PROGRAM PRG_LD


VAR
    // 数据表格式
 

    // 连接到数据库
 

    // 插入新行
 

    // 查询现有数据
 

    // 更新现有数据
 


stTableSchema        : ST_ProdColumnName;;

FB_ConnSQLServer_0   : FB_ConnSQLServer;;

stNewProd            : ST_ProdEntry;;

FB_InsertSQLServer_0 : FB_InsertSQLServer;;

stQueryProd          : ST_ProdEntry;;

FB_QuerySQLServer_0  : FB_QuerySQLServer;;

stUpdateProd         : ST_ProdEntry;;

FB_UpdateSQLServer_0 : FB_UpdateSQLServer;;

    END_VAR

END_PROGRAM

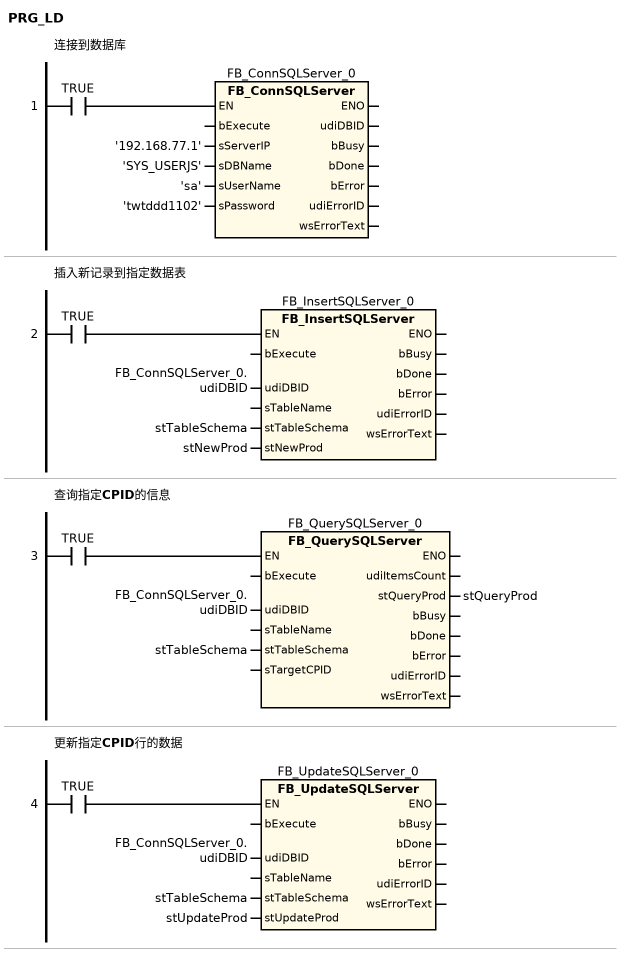
// NETWORK 1: 连接到数据库
FB_ConnSQLServer_0(
    sServerIP := '192.168.77.1',
    sDBName := 'SYS_USERJS',
    sUserName := 'sa',
    sPassword := 'twtddd1102'); // FB_ConnSQLServer

// NETWORK 2: 插入新记录到指定数据表
FB_InsertSQLServer_0(
    udiDBID := FB_ConnSQLServer_0.udiDBID,
    stTableSchema := stTableSchema,
    stNewProd := stNewProd); // FB_InsertSQLServer

// NETWORK 3: 查询指定CPID的信息
FB_QuerySQLServer_0(
    udiDBID := FB_ConnSQLServer_0.udiDBID,
    stTableSchema := stTableSchema,
    stQueryProd => stQueryProd); // FB_QuerySQLServer

// NETWORK 4: 更新指定CPID行的数据
FB_UpdateSQLServer_0(
    udiDBID := FB_ConnSQLServer_0.udiDBID,
    stTableSchema := stTableSchema,
    stUpdateProd := stUpdateProd); // FB_UpdateSQLServer

END_PROGRAM

(* stored: Version 1.1.0.1, ProductVersion 3.1.4024.16
   POU PRG_LD: Id {c4176d62-33bc-4c25-bb2c-7a9773f7c879}, SpecialFunc None *)
